PROGRAM MAIN
VAR
END_VAR

END_PROGRAM

(* stored: Version 1.1.0.1
   POU MAIN: Id {1fa6bdac-2231-4a31-95f5-dde1d508cce4} *)
